(* IEC 61131-3 sources: ATCMcontrol_Engineering/src/COM/softing/fc/AddOns/Softing/4CPCTarget/Libs/ATCM_IEC1131_3/table_29, 17 files *)

(* ---- concat.st ---- *)
FUNCTION CONCAT : ANY_STRING
VAR_INPUT
    IN1 : ANY_STRING;
END_VAR
VAR_IN_EXT
    IN2 : ANY_STRING;
END_VAR

overload() inline {@+}

END_FUNCTION

(* ---- delete.st ---- *)
FUNCTION DELETE : ANY_STRING
VAR_INPUT
    IN : ANY_STRING;
    L : ANY_INT;
    P : ANY_INT;
END_VAR

overload STRING(STRING,INT,INT)
    inline{ STDLIB(DeleteString_int)}

overload STRING(STRING,DINT,DINT)
    inline{
        %res
        %2
        dint_to_int
        %3
        dint_to_int
        %1
        calfsys #DeleteString_int
		leave 8
        }

(*
overload STRING(STRING,LINT,LINT)
    inline{
        %res
        %2
        lint_to_int
        %3
        lint_to_int
        %1
        calfsys #DeleteString_int
	leave 12
        }

overload STRING(STRING,SINT,SINT)
    inline{
        %res
        %2
        sint_to_int
        %3
        sint_to_int
        %1
        calfsys #DeleteString_int
	leave 12
        }
*)

END_FUNCTION

(* ---- delete_dint.st ---- *)
FUNCTION DELETE_DINT : ANY_STRING
VAR_INPUT
    IN : ANY_STRING;
    L  : DINT;
    P  : DINT;
END_VAR

overload() inline{Utils.deleteString(%1,%2,%3)}

END_FUNCTION

(* ---- find.st ---- *)
FUNCTION FIND : ANY_INT
VAR_INPUT
    IN1 : ANY_STRING;
    IN2 : ANY_STRING;
END_VAR

overload INT(STRING,STRING)
    inline{ STDLIB(FindString_int) }

overload DINT(STRING,STRING)
    inline{
        %res
        dint_to_int
        %2
        %1
        calfsys #FindString_int
		leave 8
		int_to_dint
        }

(*
overload LINT(STRING,STRING)
    inline{
        %res
        lint_to_int
        %2
        %1
        calfsys #FindString_int
	leave 10
        }

overload SINT(STRING,STRING)
    inline{
        %res
        sint_to_int
        %2
        %1
        calfsys #FindString_int
	leave 10
        }
*)

END_FUNCTION

(* ---- find_dint.st ---- *)
FUNCTION FIND_DINT : DINT
VAR_INPUT
    IN1 : ANY_STRING;
    IN2 : ANY_STRING;
END_VAR

overload() inline{%1.indexOf(%2)+1}

END_FUNCTION

(* ---- insert.st ---- *)
FUNCTION INSERT : ANY_STRING
VAR_INPUT
    IN1 : ANY_STRING;
    IN2 : ANY_STRING;
    P : ANY_INT;
END_VAR

overload STRING(STRING,STRING,INT)
    inline{ STDLIB(InsertString_int)}

overload STRING(STRING,STRING,DINT)
    inline{
        %res
        %3
        dint_to_int
        %2
        %1
        calfsys #InsertString_int
		leave 10
        }

(*
overload STRING(STRING,STRING,LINT)
    inline{
        %res
        %3
        lint_to_int
        %2
        %1
        calfsys #InsertString_int
	leave 14
        }

overload STRING(STRING,STRING,SINT)
    inline{
        %res
        %3
        sint_to_int
        %2
        %1
        calfsys #InsertString_int
	leave 14
        }
*)

END_FUNCTION

(* ---- insert_dint.st ---- *)
FUNCTION INSERT_DINT : ANY_STRING
VAR_INPUT
    IN1 : ANY_STRING;
    IN2 : ANY_STRING;
    P   : DINT;
END_VAR

overload() inline{Utils.insertString(%1,%2,%3)}

END_FUNCTION

(* ---- left.st ---- *)
FUNCTION LEFT : ANY_STRING
VAR_INPUT
    IN : ANY_STRING;
    L : ANY_INT;
END_VAR

overload STRING(STRING,INT)
    inline{ STDLIB(LeftString_int) }

overload STRING(STRING,DINT)
    inline{
        %res
        %2
        dint_to_int
        %1
        calfsys #LeftString_int
		leave 6
        }

(*
overload STRING(STRING,LINT)
    inline{
        %res
        %2
        lint_to_int
        %1
        calfsys #LeftString_int
        leave 10
        }

overload STRING(STRING,SINT)
    inline{
        %res
        %2
        sint_to_int
        %1
        calfsys #LeftString_int
        leave 10
        }
*)

END_FUNCTION

(* ---- left_dint.st ---- *)
FUNCTION LEFT_DINT : ANY_STRING
VAR_INPUT
    IN : ANY_STRING;
    L  : DINT;
END_VAR

overload() inline{Utils.leftString(%1,%2)}

END_FUNCTION

(* ---- len.st ---- *)
FUNCTION LEN : ANY_INT
VAR_INPUT
    IN : STRING;
END_VAR

overload INT(STRING) inline { STDLIB(strlen_int) }
overload DINT(STRING) inline
{
	%res
	%1
    calfsys #strlen_int %leave
    int_to_dint
}

END_FUNCTION

(* ---- len_dint.st ---- *)
FUNCTION LEN_DINT : DINT
VAR_INPUT
    IN : ANY_STRING;
END_VAR

overload() inline{%1.length()}

END_FUNCTION

(* ---- mid.st ---- *)
FUNCTION MID : ANY_STRING
VAR_INPUT
    IN : ANY_STRING;
    L : ANY_INT;
    P : ANY_INT;
END_VAR

overload STRING(STRING,INT,INT)
    inline{ STDLIB(MidString_int) }

overload STRING(STRING,DINT,DINT)
    inline{
        %res
        %2
        dint_to_int
        %3
        dint_to_int
	    %1
        calfsys #MidString_int
		leave  8
        }

(*
overload STRING(STRING,LINT,LINT)
    inline{
        %res
        %2
        lint_to_int
        %3
        lint_to_int
	%1
        calfsys #MidString_int
        leave 12
        }

overload STRING(STRING,SINT,SINT)
    inline{
        %res
        %2
        sint_to_int
        %3
        sint_to_int
	%1
        calfsys #MidString_int
        leave 12
        }
*)

END_FUNCTION

(* ---- mid_dint.st ---- *)
(*[[
    UserURL= "ATCM:MID_DINT.htm"
]]*)

FUNCTION MID_DINT : ANY_STRING
VAR_INPUT
    IN : ANY_STRING;
    L  : DINT;
    P  : DINT;
END_VAR

overload() inline{Utils.midString(%1,%2,%3)}

END_FUNCTION

(* ---- replace.st ---- *)
FUNCTION REPLACE : ANY_STRING
VAR_INPUT
    IN1 : ANY_STRING;
    IN2 : ANY_STRING;
    L : ANY_INT;
    P : ANY_INT;
END_VAR

overload STRING(STRING,STRING,INT,INT)
    inline{ STDLIB(ReplaceString_int) }

overload STRING(STRING,STRING,DINT,DINT)
    inline{
        %res
        %3
        dint_to_int
        %4
        dint_to_int
        %2
        %1
        calfsys #ReplaceString_int
		leave  12
        }

(*
overload STRING(STRING,STRING,LINT,LINT)
    inline{
        %res
        %3
        lint_to_int
        %4
        lint_to_int
        %2
        %1
        calfsys #ReplaceString_int
	leave 16
        }

overload STRING(STRING,STRING,SINT,SINT)
    inline{
        %res
        %3
        sint_to_int
        %4
        sint_to_int
        %2
        %1
        calfsys #ReplaceString_int
	leave 16
        }
*)

END_FUNCTION

(* ---- replace_dint.st ---- *)
(*[[
    UserURL= "ATCM:REPLACE_DINT.htm"
]]*)

FUNCTION REPLACE_DINT : ANY_STRING
VAR_INPUT
    IN1 : ANY_STRING;
    IN2 : ANY_STRING;
    L   : DINT;
    P   : DINT;
END_VAR

overload() inline{Utils.replaceString(%1,%2,%3,%4)}

END_FUNCTION

(* ---- right.st ---- *)
FUNCTION RIGHT : ANY_STRING
VAR_INPUT
    IN : ANY_STRING;
    L : ANY_INT;
END_VAR

overload STRING(STRING,INT)
    inline{ STDLIB(RightString_int) }

overload STRING(STRING,DINT)
    inline{
        %res
        %2
        dint_to_int
        %1
        calfsys #RightString_int
		leave  6
        }

(*
overload STRING(STRING,LINT)
    inline{
        %res
        %2
        lint_to_int
        %1
        calfsys #RightString_int
	leave 10
        }

overload STRING(STRING,SINT)
    inline{
        %res
        %2
        sint_to_int
        %1
        calfsys #RightString_int
	leave 10
        }
*)

END_FUNCTION

(* ---- right_dint.st ---- *)
FUNCTION RIGHT_DINT : ANY_STRING
VAR_INPUT
    IN : ANY_STRING;
    L  : DINT;
END_VAR

overload() inline{Utils.rightString(%1,%2)}

END_FUNCTION
